// TwinCAT 3 PLC project DCS_offline_var_test
// ProgramVersion: 3.1.4023.0
// libraries:
//   Tc2_Standard, * (Beckhoff Automation GmbH)
//   Tc2_System, * (Beckhoff Automation GmbH)
//   Tc3_Module, * (Beckhoff Automation GmbH)
// project tree:
//   GVLs/ GVL_RESD.TcGVL, GVL_ROB.TcGVL
//   / PlcTask.TcTTO
//   POUs/ MAIN.TcPOU
// real-time tasks:
//   TASK PlcTask: cycle T#10ms, priority 20, ADS port 350

CONFIGURATION DCS_offline_var_test
    RESOURCE PLC ON TwinCAT3
        TASK PlcTask(INTERVAL := T#10ms, PRIORITY := 20);
        PROGRAM MAIN WITH PlcTask : MAIN;
    END_RESOURCE
END_CONFIGURATION

// ---- GVLs/GVL_RESD.TcGVL
{attribute 'qualified_only'}
// ***********************************************************************************
//
// Müller-steinag Gruppe, Kandergrien Einigen, CH-3646 Bern
// ETH Zurich, Building Hin E26, Laura-Hezner-Weg 7, CH-8093 Zürich
// 
// ***********************************************************************************
// 
// PROJECT     :  A061 Digital Casting System 
// FUNCTION    :  Global Proninet Varable with robot
// AUTHOR      :  Weiting Chen
// EMAIL       :  chenw@usi.ch
// Copyright   :  USI Mendrisio; ETH Zürich; Müller-steinag Gruppe (CH) 2023
//
// **************S*********************************************************************

VAR_GLOBAL
	
CONCRETE_CONTROLLER: STRING := 'MIXER';//***********************************************************
b_Operate_mode_manual : BOOL;
b_Operate_mode_laptop : BOOL; 	
b_Operate_mode_robot : BOOL; 
b_Concrete_Controller_enable : BOOL;
b_Concrete_Controller_reset : BOOL;
b_Concrete_Controller_power_on : BOOL; 
n_Concrete_Controller_current_mode : INT;

MIXER: STRING := 'MIXER';//***********************************************************
// Inline Mixer
// input 		
b_MI1_set_run : BOOL;								// POWER ON *****
b_Ml1_Enable : BOOL;
n_MI1_set_speed : REAL;								// [0 rpm to 120 rpm]
b_MI1_set_curved_speed_mode_on: BOOL;				// Curved Speed Mode

// output 
b_MI1_Is_Run:BOOL;
b_MI1_Is_ready : BOOL;
n_MI1_status_SpeedM1 : INT;
n_MI1_status_SpeedM2 : INT;
f_Status_Torque_Motor_1 : REAL;
f_Status_Torque_Motor_2 : REAL;
f_MI1_status_temperature_funnel_outlet : REAL; 		
f_MI1_status_Pressure_funnel_inlet : REAL; 	
f_MI1_status_temperature_motor_1 : REAL; 			 
f_MI1_status_temperature_motor_2 : REAL; 
f_MI1_Override_Max_Speed : REAL := 120;				// [rpm]

CONCRETE_PUMP: STRING := 'CONCRETE_PUMP';
// Concrete Pump
// input
b_Concrete_Pump_Power_On: BOOL;						
b_Concrete_Pump_Forward_On: BOOL;					// Forward ON
b_Concrete_Pump_Backward_On: BOOL;					// X

b_Concrete_Pump_Flush_On: BOOL;						// FLUSH MODE ON 
n_Concrete_Pump_Flush_Flowrate: REAL;				// READ [l/min]

b_Concrete_Pump_Check_On: BOOL;						// CHECK MODE ON 
f_Concrete_Pump_Check_Flowrate: REAL; 				// [ O tp 24 l/min]
n_Concrete_Pump_Check_Duration: INT := 15; 			// [s]

f_Concrete_Pump_Set_Flowrate: REAL; 				// [0 to 24 l/min]
f_Concrete_Pump_dosing_volume: REAL := 0.32;		// calibrated 230926 WT
n_Concrete_Pump_Max_Speed : INT := 75;
n_Concrete_Pump_Set_Speed: INT;						// WRITE VALUE From 0 to 75 [rpm] 

b_CP1_is_run : BOOL;
b_CP1_is_ready : BOOL;
b_CP1_power_on :BOOL;
b_CP1_safety_grid_on : BOOL;
b_CP1_drive_error :BOOL;
f_CP1_status_temperature_concrete_fresh : REAL; // [°C]
f_CP1_status_temperature_Concrete_pump : REAL; // [°C] 
f_CP1_status_pressure_Concrete_pump: REAL; // [bar]


//f_Concrete_Pump_Density: REAL;					// [g/ml]
//f_Concrete_Pump_Check_Mass: REAL;           		// [g]

Admixture_Pump_1: STRING := 'Admixture Pump (AP1)';

b_Admixture_Pump_Power_On : BOOL;  					// Power On
b_Admixture_Pump_Set_Run : BOOL;  					// Set Run 
b_Admixture_Pump_Flush_On: BOOL;					// FLUSH MODE ON 
f_Admixture_Pump_Flush_Flowrate: REAL;				// READ 
b_Admixture_Pump_Check_On: BOOL;					// CHECK MODE ON 
f_Admixture_Pump_Check_Flowrate: REAL;				// READ 
n_Admixture_Pump_Check_Duration: INT := 60; 		// [s]
n_Admixture_Pump_Max_Flowrate :INT  := 637;		//calibrated 2402 WT
f_Admixture_Pump_Set_Flowrate: REAL;         		// 0 to 637 [ml/min] 
f_Admixture_Pump_dosing_factor: REAL := 1;			//only for scaled

//f_Admixture_Pump_1_Density: REAL;          // [g/ml]
//f_Admixture_Pump_1_Mass: REAL;             // [g]

b_Admixture_Pump_is_run : BOOL;
b_Admixture_Pump_is_ready : BOOL;
b_Admixture_Pump_no_error : BOOL;

//
Sup_Admixture_Pump_1: STRING := 'Admixture Pump (SP1)'; //***************************


b_Sup_Admixture_Pump_Power_On : BOOL;  					// Power On
b_Sup_Admixture_Pump_Set_Run: BOOL;  					// Set Run 

b_Sup_Admixture_Pump_Flush_On: BOOL;				// FLUSH MODE ON 
f_Sup_Admixture_Pump_Flush_Flowrate: REAL;
b_Sup_Admixture_Pump_Check_On: BOOL;				// CHECK MODE ON 
f_Sup_Admixture_Pump_Check_Flowrate: REAL;
n_Sup_Admixture_Pump_Check_Duration: INT := 60; 	// [s];
n_Sup_Admixture_Pump_Max_Flowrate:INT := 138; 		//[ml/min]

f_Sup_Admixture_Pump_Set_Flowrate: REAL;         	// 0 to 138[ml/min]
f_Sup_Admixture_Pump_dosing_factor:REAL:=1; //only for scaled

//f_Admixture_Pump_2_Density: REAL;          // [g/ml]
//f_Admixture_Pump_2_Mass: REAL;             // [g]

b_Sup_Admixture_Pump_is_run : BOOL;
b_Sup_Admixture_Pump_is_ready : BOOL;
b_Sup_Admixture_Pump_no_error : BOOL;
END_VAR

// ---- GVLs/GVL_ROB.TcGVL
{attribute 'qualified_only'}
// ***********************************************************************************
//
// Müller-steinag Gruppe, Kandergrien Einigen, CH-3646 Bern
// ETH Zurich, Building Hin E26, Laura-Hezner-Weg 7, CH-8093 Zürich
// 
// ***********************************************************************************
// 
// PROJECT     :  A061 Digital Casting System 
// FUNCTION    :  Global Proninet Varable with robot
// AUTHOR      :  Weiting Chen
// EMAIL       :  chenw@usi.ch
// Copyright   :  USI Mendrisio; ETH Zürich; Müller-steinag Gruppe (CH) 2023
//
// ************************************************************************************

VAR_GLOBAL
	//output to robot digital input (DI) ; input from robot digital output(DO)
	
	//UINT type as 16bit ranged -32767 to 32767 (Here, the number is scaled by 1000
	
	//Concrete Controller
	ib_spare : BOOL;
	in_spare : INT;
	
	ib_CC1_enable : BOOL;
	ib_CC1_reset : BOOL;
	
	ob_mode_manual : BOOL;
	ob_mode_laptop : BOOL; 	
	ob_mode_robot : BOOL; 
	on_current_mode : INT; //index use no scale.
	ob_CC1_power_on : BOOL; 
	
	//Inline Mixer (MI1)  				
	ib_MI1_set_run : BOOL;
	ib_Ml1_enable : BOOL;
	ib_MI1_set_rest : BOOL;				 
	in_MI1_set_speed : UINT;								// [0 rpm to 120 rpm]
	ib_MI1_set_curved_speed_mode_on : BOOL;
	
	ob_MI1_is_run : BOOL;
	ob_MI1_is_ready : BOOL;
	
	on_MI1_status_speed_motor_1 : INT;				 	// [rpm]
	on_MI1_status_Speed_motor_2 : INT;					// [rpm]
	on_MI1_status_torque_motor_1 : REAL;					// [Nm]
	on_MI1_status_torque_motor_2 : REAL;					// [Nm]
	
	on_MI1_status_temperature_funnel_outlet : REAL; 		// [°C] 
	on_MI1_status_pressure_funnel_inlet : REAL; 			// [bar]
	on_MI1_status_temperature_motor_1 : REAL; 			// [°C] 
	on_MI1_status_temperature_motor_2 : REAL; 			// [°C] 
	
	
	//Concrete pump (CP1)  
	//ib_CP1_run: BOOL;					// NOT USE NOW
	ib_CP1_forward_on: BOOL;			    
	ib_CP1_backward_on: BOOL;			// 241219 Backward is not working from the conctroller
	in_CP1_set_flowrate: UINT; 			// 0 to 24 [l/min]
	in_CP1_set_speed: UINT;				// 0 to 75 [rpm] 
	in_CP1_set_dosing_volume: UINT;		// scale to 0 to 100 | calibration in 230926 WT 0.32
	
	ib_CP1_check_on: BOOL;			 
	in_CP1_set_check_Flowrate: UINT; 	// [l/min]
	t_CP1_set_check_duration: TIME;		//  T#1d2h30m40s500ms
	in_CP1_concrete_density: UINT;		// [g/ml]
	in_CP1_concrete_mass: UINT;          // [g]
	
	ib_CP1_flush_on: BOOL;				
	in_CP1_set_flush_flowrate: UINT;		// [l/min]
	
	on_CP1_status_temperature_concrete_fresh : REAL; // [°C]
	on_CP1_status_temperature_concrete_pump : REAL; // [°C] 
	on_CP1_status_pressure_concrete_pump: REAL; // [ bar
	
	ob_CP1_is_run : BOOL;
	ob_CP1_is_ready : BOOL;
	ob_CP1_power_on : BOOL;
	ob_CP1_safety_grid_on : BOOL;
	ob_CP1_drive_error :BOOL;
	

	
	
	// Admixture pump, High dosage ViscoTech Pump
	ib_AP1_power_on: BOOL; 
	ib_AP1_set_run: BOOL; 
	in_AP1_set_flowrate: UINT;         		// [ml/min] 
	in_AP1_set_dosing_factor: UINT;          // Set default 1
	
	ib_AP1_check_on: BOOL;			
	in_AP1_set_check_flowrate: UINT;
	t_AP1_set_check_duration: TIME;// T#1d2h30m40s500ms
	in_AP1_material_density: UINT;          // [g/ml]
	in_AP1_material_mass: UINT;             // [g]
	
	ib_AP1_flush_on: BOOL;			 
	in_AP1_set_flush_flowrate: UINT;	  // [ml/min] 
	
	ob_AP1_is_run : BOOL;
	ob_AP1_is_ready : BOOL;

	ob_AP1_no_error : BOOL;
	on_AP1_max_flowrate: UINT:=637;			// [ml/min] 	
	
	// Admixture pump, Low dosage ViscoTech Pump 
	ib_SP1_power_on: BOOL;
	ib_SP1_set_run: BOOL;
	in_SP1_set_flowrate: UINT;         // [ml/min]
	in_SP1_dosing_factor:UINT;       
	
	ib_SP1_set_check_on: BOOL;			 
	in_SP1_set_check_flowrate: UINT;	  // [ml/min] 
	t_SP1_Check_Duration: TIME ;       // T#1d2h30m40s500ms
	in_SP1_material_density: UINT;     // [g/ml]
	in_SP1_material_mass: UINT;        // [g]
	
	ib_SP1_flush_on: BOOL;			 
	in_SP1_flush_flowrate: UINT;	  // [ml/min] 
	
	ob_SP1_is_run:BOOL;
	ob_SP1_is_ready : BOOL;
	ob_SP1_no_error : BOOL;
	on_SP1_max_flowrate:UINT := 138;		  // [ml/min] 
END_VAR

// ---- POUs/MAIN.TcPOU
PROGRAM MAIN
VAR
END_VAR

END_PROGRAM
